Yaskawa INFORM job: LINDSAT.JBI

/JOB
//NAME LINDSAT
//POS
///NPOS 3,0,0,0
///TOOL 0
///PULSE
C000=33,44679,-65436,295,-3982,-2624
C001=33,49671,-53532,295,1702,-2624
C002=705,42711,-30636,379,1422,-2540
//INST
///DATE 2014/11/01 22:56
///ATTR 0,0,0,0,0,0,0,0,0,0,0,0,0,1,0,0
///FRAME BASE
NOP
*1
MOVJ C000 VJ=25.00 CONT
PAUSE
MOVJ C001 VJ=100.00 CONT
MOVJ C002 VJ=100.00 CONT
JUMP *1
END
